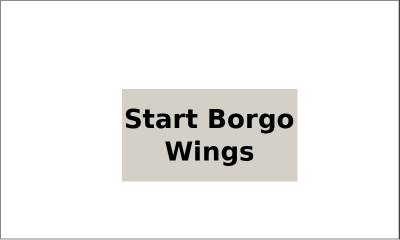
VISUALIZATION V_StartBorgoWings  // 400x240
VAR_IN_OUT
	HMI : ST_PackMLBaseModule_HMI;
END_VAR
    RoundedRectangle (0,-1 400x240)
    RoundedRectangle (122,89 175x92), "Start Borgo Wings"
        OnMouseClick: execute { HMI.Command.State := E_PMLCommand.ePMLCommand_Start; }
END_VISUALIZATION

(* stored: Version 1.1.0.1, ProductVersion 3.1.4024.15
   Visu V_StartBorgoWings: Id {efad271e-12d1-4fb0-b506-e59d88a07246} *)
